// TwinCAT 3 PLC project PLC
// ProgramVersion: 3.1.4022.3
// libraries:
//   Tc2_Standard, * (Beckhoff Automation GmbH)
//   Tc2_System, * (Beckhoff Automation GmbH)
//   Tc3_Module, * (Beckhoff Automation GmbH)
// project tree:
//   DUTs/ DAU.TcDUT
//   GVLs/ GVL_DUA.TcGVL
//   / PlcTask.TcTTO
//   POUs/Commands/ I_Command.TcIO
//   POUs/ FB_CtrlgxParser.TcPOU, MAIN.TcPOU
//   POUs/Invoker/ FB_Invoke.TcPOU
//   POUs/Receivers/ FB_DAU.TcPOU
// real-time tasks:
//   TASK PlcTask: cycle T#10ms, priority 20, ADS port 350
// I/O:
//   DEVICE Device 1 (EtherCAT), AmsNetId 192.168.2.38.2.1
//     Box 1 (EPP2318-0001) [EPP2318-0001 4 Ch. Dig. In, 10µs, 4 Ch. Dig. Out 24V, 0,5A, M8]

CONFIGURATION PLC
    RESOURCE PLC ON TwinCAT3
        TASK PlcTask(INTERVAL := T#10ms, PRIORITY := 20);
        PROGRAM MAIN WITH PlcTask : MAIN;
    END_RESOURCE
END_CONFIGURATION

// ---- DUTs/DAU.TcDUT
TYPE DAU :
STRUCT
	//Divert 1 IO //
	bDivert1Extend : BOOL; //Extend Signal to Solenoid
	bDivert1Retract : BOOL; //Retract Signal to Solenoid
	bDivert1Faulted : BOOL; //Faulted Status to Line Controller
	bDivert1MissingPin : BOOL; //Missing Pin input from shoe sensor
	bDivert1SWSensor : BOOL; //SW Sensor from shoe sensor
	bDivert1GO : BOOL;  // Divert signal from Line Controller
	//Divert 2 IO //
	bDivert2Extend : BOOL;
	bDivert2Retract : BOOL;
	bDivert2Faulted : BOOL; //Faulted Status to Line Controller
	bDivert2MissingPin : BOOL; //Missing Pin input from shoe sensor
	bDivert2SWSensor : BOOL; //SW Sensor from shoe sensor
	bDivert2GO : BOOL;  // Divert signal from Line Controller
	//END
END_STRUCT
END_TYPE

// ---- GVLs/GVL_DUA.TcGVL
VAR_GLOBAL
	DAU : ARRAY [1..100] OF DAU; //Instantiate 100 DAU's  This can be made higher if we think that 1 system will ever have more than 100 DAU's
END_VAR

// ---- POUs/Commands/I_Command.TcIO
INTERFACE I_Command

METHOD Execute
END_METHOD

END_INTERFACE

// ---- POUs/MAIN.TcPOU
PROGRAM MAIN
VAR
END_VAR

END_PROGRAM

// ---- POUs/FB_CtrlgxParser.TcPOU
FUNCTION_BLOCK FB_CtrlgxParser
VAR_INPUT
END_VAR
VAR_OUTPUT
END_VAR
VAR
END_VAR
xdfsdfsd

END_FUNCTION_BLOCK

// ---- POUs/Invoker/FB_Invoke.TcPOU
FUNCTION_BLOCK FB_Invoke
VAR_INPUT
END_VAR
VAR_OUTPUT
END_VAR
VAR
END_VAR

END_FUNCTION_BLOCK

// ---- POUs/Receivers/FB_DAU.TcPOU
FUNCTION_BLOCK FB_DAU
VAR_INPUT
END_VAR
VAR_OUTPUT
END_VAR
VAR
END_VAR

METHOD PUBLIC Extend : BOOL
VAR_INPUT
END_VAR
END_METHOD

METHOD PUBLIC Init : BOOL
VAR_INPUT
END_VAR
END_METHOD

METHOD PUBLIC Retract : BOOL
VAR_INPUT
END_VAR
END_METHOD

METHOD PUBLIC TrigFault : BOOL
VAR_INPUT
END_VAR
END_METHOD

END_FUNCTION_BLOCK
